{attribute 'GeneratedUsingTerminal: EPP2339-0003-0016'}
{attribute addProperty BoxType "EPP2339-0003-0016"}
{attribute addProperty Id "DI_Inputs_Channel_1AT %I*DI_Inputs_Channel_91AC31B711DI_Inputs_Channel_2AT %I*DI_Inputs_Channel_91AC31B711DO_Outputs_Channel_1AT %Q*DO_Outputs_Channel_28AC1A9E8DO_Outputs_Channel_2AT %Q*DO_Outputs_Channel_28AC1A9E8WcStateAT %I*WcState_9091E0EB2InfoDataAT %I*InfoData_32EB74EA10"}
{attribute addProperty CRC "2998276840"}
{attribute addProperty Size "50"}
TYPE EPP2339_B2B612E8 EXTENDS EtcSlaveTerminalBase_947E5A46 :
STRUCT
	{attribute addProperty Name "DI_Inputs_Channel_1"}
	DI_Inputs_Channel_1 : DI_Inputs_Channel_91AC31B7;
	{attribute addProperty Name "DI_Inputs_Channel_2"}
	DI_Inputs_Channel_2 : DI_Inputs_Channel_91AC31B7;
	{attribute addProperty Name "DO_Outputs_Channel_1"}
	DO_Outputs_Channel_1 : DO_Outputs_Channel_28AC1A9E;
	{attribute addProperty Name "DO_Outputs_Channel_2"}
	DO_Outputs_Channel_2 : DO_Outputs_Channel_28AC1A9E;
	{attribute addProperty Name "WcState"}
	WcState : WcState_9091E0EB;
	{attribute addProperty Name "InfoData"}
	InfoData : InfoData_32EB74EA;
END_STRUCT
END_TYPE

(* stored: Version 1.2.0.0, ProductVersion 3.1.4024.9
   DUT EPP2339_B2B612E8: Id {c8e91af4-cf55-4769-bc6a-06ccfe8fdfda} *)
